TYPE DUT_SATT_Filter :
STRUCT
    {attribute 'pytmc' := '
        pv: MATERIAL
        io: input
        field: DESC Filter material name
    '}
    sFilterMaterial : STRING;

    {attribute 'pytmc' := '
        pv: THICKNESS
        io: input
        field: DESC Filter material thickness
        field: EGU um
    '}
    fFilterThickness_um : LREAL;

    {attribute 'pytmc' := '
        pv: TRANSMISSION
        io: input
        field: DESC Current transmission value
    '}
    fTransmission : LREAL;

END_STRUCT
END_TYPE

(* stored: Version 1.1.0.1, ProductVersion 3.1.4022.18
   DUT DUT_SATT_Filter: Id {3bb2cd4a-447e-0bc9-0e20-a4850e5ce007} *)
